E_OpStep.VMCAS_VENTING: // Venting, increase opening by X% every 2 miniutes, until at atmosphere
    DREAM_ROUGH2_VFV_02.M_SetControlMode(E_VCN.ManualControl); // set manual mode for VFV valve
    DREAM_ROUGH2_VFV_03.M_SetControlMode(E_VCN.ManualControl); // set manual mode for VFV valve
    // Verify ATM_PRESS_ERR_RNG value with testing
    IF NOT (ABS(ATM_PRESS - DREAM_DP1_GPI_01.PG.rPRESS) <= ATM_PRESS_ERR_RNG)
        AND NOT (ABS(ATM_PRESS - DREAM_MC_GPI_01.PG.rPRESS) <= ATM_PRESS_ERR_RNG)
        AND NOT (ABS(ATM_PRESS - DREAM_ROUGH2_GPI_02.PG.rPRESS) <= ATM_PRESS_ERR_RNG)
        AND NOT (ABS(ATM_PRESS - DREAM_ROUGH2_GPI_03.PG.rPRESS) <= ATM_PRESS_ERR_RNG)
    THEN
        M_RunTimeoutTimer(VENTING_CYCLE);
        M_SetMessage('Venting Started');
        // Add check if serial communication is ok. If not ok we should only stick to change open position by 1% until venting completed?
        // I think we should add range here for the speed 1-5 Hz? I think sometimes speed doesn't go all the way to 0 Hz, verify with testing
        IF M_TimeoutExpired() THEN
            M_ResetTimeoutTimer(); // Reset timer for next 2 min venting cycle
            IF (NOT (DREAM_DP1_PTM_01.iq_stPTM.i_diCurSpd < 1) OR fbSerialLineControl_DREAM_DP1_PTM_01.Error)
                AND (NOT (DREAM_DP2_PTM_01.iq_stPTM.i_diCurSpd < 1) OR fbSerialLineControl_DREAM_DP2_PTM_01.Error)
                AND (NOT (DREAM_DP3_PTM_01.iq_stPTM.i_diCurSpd < 1) OR fbSerialLineControl_DREAM_DP3_PTM_01.Error)
                AND (NOT (DREAM_MC_PTM_01.iq_stPTM.i_diCurSpd < 1) OR fbSerialLineControl_DREAM_MC_PTM_01.Error)
                AND (NOT (DREAM_MC_PTM_02.iq_stPTM.i_diCurSpd < 1) OR fbSerialLineControl_DREAM_MC_PTM_01.Error)
                AND (NOT (DREAM_CAT1_PTM_01.iq_stPTM.i_diCurSpd < 1) OR fbSerialLineControl_DREAM_CAT1_PTM_01.Error)
                AND (NOT (DREAM_CAT2_PTM_01.iq_stPTM.i_diCurSpd < 1) OR fbSerialLineControl_DREAM_CAT2_PTM_01.Error)
                AND (NOT (DREAM_ROUGH2_PTM_01.iq_stPTM.i_diCurSpd < 1) OR fbSerialLineControl_DREAM_ROUGH2_PTM_01.Error)
                AND (NOT (DREAM_ROUGH2_PTM_02.iq_stPTM.i_diCurSpd < 1) OR fbSerialLineControl_DREAM_ROUGH2_PTM_02.Error)
            THEN
                IF fRough2VFV2Position < VFV_MAX_POSITION THEN
                    fRough2VFV2Position := fRough2VFV2Position + VFV_POSITION_STEP; // every 2 min increase open positon for 1% while pumps above 1 HZ
                ELSE
                    fRough2VFV2Position := VFV_MAX_POSITION;
                END_IF

                IF fRough2VFV3Position < VFV_MAX_POSITION THEN
                    fRough2VFV3Position := fRough2VFV3Position + VFV_POSITION_STEP; // every 2 min increase open positon for 1% while pumps above 1 HZ
                ELSE
                    fRough2VFV3Position := VFV_MAX_POSITION;
                END_IF
            ELSE
                fRough2VFV2Position := VFV_MAX_POSITION; // open venting valve to max postion when pump speed reached below 1Hz
                fRough2VFV3Position := VFV_MAX_POSITION; // open venting valve to max postion when pump speed reached below 1Hz
            END_IF
        END_IF
    ELSE
        M_SetMessage('Venting completed');
        M_ResetTimeoutTimer();
        eStep := E_OpStep.VMCAS_FINISH;
    END_IF

    DREAM_ROUGH2_VFV_02.M_SetReqPosition(fRough2VFV2Position); // set venting valve position
    DREAM_ROUGH2_VFV_03.M_SetReqPosition(fRough2VFV3Position); // set venting valve position

E_OpStep.VMCAS_FINISH: // Finish procedure, close venting valves, reset set points for all valves, pumps etc.
    DREAM_ROUGH2_VFV_02.M_SetControlMode(E_VCN.CloseValve);
    DREAM_ROUGH2_VFV_03.M_SetControlMode(E_VCN.CloseValve);
    // Reset vent valve postions
    fRough2VFV2Position := 0;
    fRough2VFV3Position := 0;

    // Set the at vacuum interlocks so user can't just start opening the valves
    DREAM_ROUGH2_VRC_01.M_SetAtVacSP(VALVE_INTERLOCK_SP);
    DREAM_ROUGH2_VRC_02.M_SetAtVacSP(VALVE_INTERLOCK_SP);

    // Set the at vacuum interlocks so user can't just start turning on pumps
    DREAM_DP1_PTM_01.M_SetBackingSP(PTM_INTERLOCK_SP);
    DREAM_DP2_PTM_01.M_SetBackingSP(PTM_INTERLOCK_SP);
    DREAM_DP3_PTM_01.M_SetBackingSP(PTM_INTERLOCK_SP);
    DREAM_MC_PTM_01.M_SetBackingSP(PTM_INTERLOCK_SP);
    DREAM_MC_PTM_02.M_SetBackingSP(PTM_INTERLOCK_SP);
    DREAM_CAT1_PTM_01.M_SetBackingSP(PTM_INTERLOCK_SP);
    DREAM_CAT2_PTM_01.M_SetBackingSP(PTM_INTERLOCK_SP);
    DREAM_ROUGH2_PTM_01.M_SetBackingSP(PTM_INTERLOCK_SP);
    DREAM_ROUGH2_PTM_02.M_SetBackingSP(PTM_INTERLOCK_SP);

    // Remove command to close beamline window valves
    GVL_PLC_Interface.bCLOSE_TMO_MR5K4_VWC := FALSE;
    GVL_PLC_Interface.bCLOSE_TMO_TM2K4_VWC := FALSE;

    M_Finish();

ELSE
    M_FatalError('Operation is in invalid state');
END_CASE

END_FUNCTION_BLOCK

// ---- POUs/Automation/Abstracts/FB_Operation.TcPOU
FUNCTION_BLOCK FB_Operation
VAR_INPUT
    i_bExecute : BOOL; // Flag that indicates the operation should be ran
    i_bCancel : BOOL; // Cancel operation input signal
END_VAR
VAR_IN_OUT
    iq_sMessageBuffer : STRING(EPICS_STRING_SIZE); // Human readable description of the current step
END_VAR
VAR_OUTPUT
    q_bError : BOOL; // Whether a fatal error was encountered
    q_bBusy : BOOL; // Whether the current operation is executing
END_VAR
VAR
    bCancel : BOOL; // Saved cancel operation signal
    bDeferCancel : BOOL; // Setting to True prevents operation from being immediatly cancelled with i_bCancel. Resets to FALSE after operation finishes
    eStep : E_OpStep := E_OpStep.IDLE; // The current operation step
    fbTimeoutTimer : TON; // Timer used for tracking operation timeouts
END_VAR

IF eStep = E_OpStep.IDLE AND i_bExecute = TRUE THEN
    // Start operation
    eStep := E_OpStep.START;
    q_bBusy := TRUE;
    M_ResetError();
END_IF

(* Save the input i_bCancel signal since cancelling can take multiple cycles *)
IF i_bCancel THEN
    bCancel := TRUE;
END_IF

(* Allow operation to be cancelled from an input signal.
 The cancel input signal can be deferred by the operation if the
 operation is not at a good point to finish cancelling. *)
IF eStep <> E_OpStep.IDLE AND NOT bDeferCancel AND bCancel THEN
    M_Cancel();
END_IF

IF M_TimeoutExpired() THEN // If a timeout has expired, trigger a fatal error
    M_FatalError('Timeout expired');
END_IF

METHOD PROTECTED M_Cancel
VAR_INPUT
END_VAR
M_ResetTimeoutTimer();
M_SetMessage('Operation canceled');
eStep := E_OpStep.IDLE;
q_bBusy := FALSE;
bCancel := FALSE;
M_DeferCancel(FALSE);
END_METHOD

// Defer cancel signals until a later time
METHOD PROTECTED M_DeferCancel
VAR_INPUT
    i_bDefer : BOOL;
END_VAR
bDeferCancel := i_bDefer;
END_METHOD

METHOD PROTECTED M_FatalError
VAR_INPUT
    i_ErrorMessage : STRING;
END_VAR
M_ResetTimeoutTimer();
M_SetMessage(i_ErrorMessage);
eStep := E_OpStep.IDLE;
q_bError := TRUE;
q_bBusy := FALSE;
bCancel := FALSE;
M_DeferCancel(FALSE);
END_METHOD

METHOD PROTECTED M_Finish
VAR_INPUT
END_VAR
M_ResetTimeoutTimer();
M_SetMessage('Operation finished');
eStep := E_OpStep.IDLE;
q_bBusy := FALSE;
bCancel := FALSE;
M_DeferCancel(FALSE);
END_METHOD

METHOD PROTECTED M_ResetError
VAR_INPUT
END_VAR
q_bError := FALSE;
END_METHOD

METHOD PROTECTED M_ResetTimeoutTimer
VAR_INPUT
END_VAR
fbTimeoutTimer(IN := FALSE);
END_METHOD

METHOD PROTECTED M_RunTimeoutTimer
VAR_INPUT
    i_tTime : TIME; // How long the timer should run before signalling a timeout
END_VAR
fbTimeoutTimer(IN := TRUE, PT := i_tTime);
END_METHOD

METHOD PROTECTED M_SetMessage
VAR_INPUT
    i_sMessage : STRING(EPICS_STRING_SIZE);
END_VAR
iq_sMessageBuffer := i_sMessage;
END_METHOD

METHOD PROTECTED M_TimeoutExpired : BOOL
VAR_INPUT
END_VAR
fbTimeoutTimer(); // Advance timer
M_TimeoutExpired := fbTimeoutTimer.Q;
END_METHOD

END_FUNCTION_BLOCK

// ---- POUs/Automation/FB_AtVacuum.TcPOU
FUNCTION_BLOCK FB_AtVacuum EXTENDS FB_Operation
VAR_INPUT
END_VAR
VAR_OUTPUT
END_VAR
VAR
END_VAR

SUPER^(iq_sMessageBuffer := iq_sMessageBuffer);

CASE eStep OF
E_OpStep.IDLE: // Do nothing

E_OpStep.START: // Start monitoring main chamber vacuum
    IF NOT (F_AllPumpsRunning() AND F_PressAtVacSP()) THEN // add case if already vented to just cancel operation
        M_RunTimeoutTimer(TURBOS_NOT_RUNNING_TIMEOUT);
        M_SetMessage('Vacuum lost, 10 min timer started');
        IF M_TimeoutExpired() THEN
            M_FatalError('Vacuum not restored, venting started');
        END_IF
    ELSE
        M_ResetTimeoutTimer(); //reset timer if pump restarted or gauge restarted and vaccum ok
        M_SetMessage('MC Vacuum OK');
    END_IF

ELSE
    M_FatalError('Operation is in invalid state');
END_CASE

END_FUNCTION_BLOCK

// ---- POUs/Functions/F_AllPumpsRunning.TcPOU
FUNCTION F_AllPumpsRunning : BOOL
VAR_INPUT
END_VAR
VAR
END_VAR

// Pump running state verifys that iq_stPtm.i_xAtSpd AND iq_stPtm.q_RunDO are TRUE
F_AllPumpsRunning := //DREAM_NC_PTM_01.iq_stPTM.eState = E_PumpState.pumpRUNNING AND
                     //DREAM_NC_PTM_02.iq_stPTM.eState = E_PumpState.pumpRUNNING AND
                     DREAM_DP1_PTM_01.iq_stPTM.eState = E_PumpState.pumpRUNNING AND
                     DREAM_DP2_PTM_01.iq_stPTM.eState = E_PumpState.pumpRUNNING AND
                     DREAM_DP3_PTM_01.iq_stPTM.eState = E_PumpState.pumpRUNNING AND
                     DREAM_MC_PTM_01.iq_stPTM.eState = E_PumpState.pumpRUNNING AND
                     DREAM_MC_PTM_02.iq_stPTM.eState = E_PumpState.pumpRUNNING AND
                     DREAM_CAT1_PTM_01.iq_stPTM.eState = E_PumpState.pumpRUNNING AND
                     DREAM_CAT2_PTM_01.iq_stPTM.eState = E_PumpState.pumpRUNNING AND
                     DREAM_ROUGH2_PTM_01.iq_stPTM.eState = E_PumpState.pumpRUNNING AND
                     DREAM_ROUGH2_PTM_02.iq_stPTM.eState = E_PumpState.pumpRUNNING;

END_FUNCTION

// ---- POUs/Functions/F_PressAtVacSP.TcPOU
FUNCTION F_PressAtVacSP : BOOL
VAR_INPUT
END_VAR
VAR
END_VAR

F_PressAtVacSP := //DREAM_NC_GCC_01.IG.rPRESS < ATVAC_INTERLOCK_SP AND DREAM_NC_GCC_01.IG.xPRESS_OK AND
                  //DREAM_DP1_GHC_01.IG.rPRESS < ATVAC_INTERLOCK_SP AND DREAM_DP1_GHC_01.IG.xPRESS_OK AND
                  //DREAM_DP2_GHC_01.IG.rPRESS < ATVAC_INTERLOCK_SP AND DREAM_DP2_GHC_01.IG.xPRESS_OK AND
                  //DREAM_DP3_GHC_01.IG.rPRESS < ATVAC_INTERLOCK_SP AND DREAM_DP3_GHC_01.IG.xPRESS_OK AND
                  //DREAM_CAT1_GHC_01.IG.rPRESS < ATVAC_INTERLOCK_SP AND DREAM_CAT1_GHC_01.IG.xPRESS_OK AND
                  //DREAM_CAT2_GHC_01.IG.rPRESS < ATVAC_INTERLOCK_SP AND DREAM_CAT2_GHC_01.IG.xPRESS_OK AND
                  GVL_VAC_GAUGES.stDREAM_MC_GAUGE.rPRESS < AT_VAC_SP AND GVL_VAC_GAUGES.stDREAM_MC_GAUGE.xPRESS_OK;
                  //GVL_VAC_GAUGES.stDREAM_MC_GHC.xAT_VAC;
                  //we could also be checking ST_VG.xAT_VAC flag and make this value changeable?

END_FUNCTION

// ---- POUs/Functions/F_IsValidStateTransition.TcPOU
FUNCTION F_IsValidStateTransition : BOOL
VAR_INPUT
    eCurrentState : E_Op;
    eNextState : E_Op;
END_VAR
VAR
END_VAR

CASE eCurrentState OF

E_Op.INIT:
    F_IsValidStateTransition := (eNextState = E_Op.STANDBY);

E_Op.STANDBY:
    F_IsValidStateTransition := (eNextState = E_Op.STANDBY) OR
                                //(eNextState = E_Op.PUMP_ALL) OR
                                //(eNextState = E_Op.PUMP_NC) OR
                                (eNextState = E_Op.VENT_MC_CAT); // OR
                                //(eNextState = E_Op.VENT_ALL) OR
                                //(eNextState = E_Op.VENT_NC) OR
                                //(eNextState = E_Op.VENT_CAT);
                                //uncomment after procedures implemented
E_Op.PUMP_ALL:
    F_IsValidStateTransition := (eNextState = E_Op.STANDBY);

E_Op.PUMP_NC:
    F_IsValidStateTransition := (eNextState = E_Op.STANDBY);

E_Op.AT_VACUUM:
    F_IsValidStateTransition := (eNextState = E_Op.VENT_MC_CAT); //OR
                                //(eNextState = E_Op.VENT_ALL) OR
                                //(eNextState = E_Op.VENT_NC) OR
                                //(eNextState = E_Op.VENT_CAT);
                                //uncomment after procedures implemented

E_Op.VENT_ALL:
    F_IsValidStateTransition := (eNextState = E_Op.STANDBY);

E_Op.VENT_NC:
    F_IsValidStateTransition := (eNextState = E_Op.STANDBY);

E_Op.VENT_MC_CAT:
    F_IsValidStateTransition := (eNextState = E_Op.STANDBY);

E_Op.VENT_CAT:
    F_IsValidStateTransition := (eNextState = E_Op.STANDBY);

ELSE
    F_IsValidStateTransition := FALSE;
END_CASE;

END_FUNCTION

// ---- POUs/PRG_COM.TcPOU
PROGRAM PRG_COM
VAR

END_VAR

(*Instanitate Serial port com function *)
fbSerialLineControl_DREAM_NC_PTM_01(
    Mode:= SERIALLINEMODE_EL6_22B,
    pComIn:= ADR(stComIn_DREAM_NC_PTM_01),
    pComOut:= ADR(stComOut_DREAM_NC_PTM_01),
    SizeComIn:= UINT_TO_INT(SIZEOF(stComIn_DREAM_NC_PTM_01)),
    TxBuffer:= SerialTXBuffer_DREAM_NC_PTM_01,
    RxBuffer:= SerialRXBuffer_DREAM_NC_PTM_01,
    Error=> ,
    ErrorID=> );

fbSerialLineControl_DREAM_NC_PTM_02(
    Mode:= SERIALLINEMODE_EL6_22B,
    pComIn:= ADR(stComIn_DREAM_NC_PTM_02),
    pComOut:= ADR(stComOut_DREAM_NC_PTM_02),
    SizeComIn:= UINT_TO_INT(SIZEOF(stComIn_DREAM_NC_PTM_02)),
    TxBuffer:= SerialTXBuffer_DREAM_NC_PTM_02,
    RxBuffer:= SerialRXBuffer_DREAM_NC_PTM_02,
    Error=> ,
    ErrorID=> );

fbSerialLineControl_DREAM_DP1_PTM_01(
    Mode:= SERIALLINEMODE_EL6_22B,
    pComIn:= ADR(stComIn_DREAM_DP1_PTM_01),
    pComOut:= ADR(stComOut_DREAM_DP1_PTM_01),
    SizeComIn:= UINT_TO_INT(SIZEOF(stComIn_DREAM_DP1_PTM_01)),
    TxBuffer:= SerialTXBuffer_DREAM_DP1_PTM_01,
    RxBuffer:= SerialRXBuffer_DREAM_DP1_PTM_01,
    Error=> ,
    ErrorID=> );

fbSerialLineControl_DREAM_DP2_PTM_01(
    Mode:= SERIALLINEMODE_EL6_22B,
    pComIn:= ADR(stComIn_DREAM_DP2_PTM_01),
    pComOut:= ADR(stComOut_DREAM_DP2_PTM_01),
    SizeComIn:= UINT_TO_INT(SIZEOF(stComIn_DREAM_DP2_PTM_01)),
    TxBuffer:= SerialTXBuffer_DREAM_DP2_PTM_01,
    RxBuffer:= SerialRXBuffer_DREAM_DP2_PTM_01,
    Error=> ,
    ErrorID=> );

fbSerialLineControl_DREAM_DP3_PTM_01(
    Mode:= SERIALLINEMODE_EL6_22B,
    pComIn:= ADR(stComIn_DREAM_DP3_PTM_01),
    pComOut:= ADR(stComOut_DREAM_DP3_PTM_01),
    SizeComIn:= UINT_TO_INT(SIZEOF(stComIn_DREAM_DP3_PTM_01)),
    TxBuffer:= SerialTXBuffer_DREAM_DP3_PTM_01,
    RxBuffer:= SerialRXBuffer_DREAM_DP3_PTM_01,
    Error=> ,
    ErrorID=> );

fbSerialLineControl_DREAM_MC_PTM_01(
    Mode:= SERIALLINEMODE_EL6_22B,
    pComIn:= ADR(stComIn_DREAM_MC_PTM_01),
    pComOut:= ADR(stComOut_DREAM_MC_PTM_01),
    SizeComIn:= UINT_TO_INT(SIZEOF(stComIn_DREAM_MC_PTM_01)),
    TxBuffer:= SerialTXBuffer_DREAM_MC_PTM_01,
    RxBuffer:= SerialRXBuffer_DREAM_MC_PTM_01,
    Error=> ,
    ErrorID=> );

fbSerialLineControl_DREAM_MC_PTM_02(
    Mode:= SERIALLINEMODE_EL6_22B,
    pComIn:= ADR(stComIn_DREAM_MC_PTM_02),
    pComOut:= ADR(stComOut_DREAM_MC_PTM_02),
    SizeComIn:= UINT_TO_INT(SIZEOF(stComIn_DREAM_MC_PTM_02)),
    TxBuffer:= SerialTXBuffer_DREAM_MC_PTM_02,
    RxBuffer:= SerialRXBuffer_DREAM_MC_PTM_02,
    Error=> ,
    ErrorID=> );

fbSerialLineControl_DREAM_CAT1_PTM_01(
    Mode:= SERIALLINEMODE_EL6_22B,
    pComIn:= ADR(stComIn_DREAM_CAT1_PTM_01),
    pComOut:= ADR(stComOut_DREAM_CAT1_PTM_01),
    SizeComIn:= UINT_TO_INT(SIZEOF(stComIn_DREAM_CAT1_PTM_01)),
    TxBuffer:= SerialTXBuffer_DREAM_CAT1_PTM_01,
    RxBuffer:= SerialRXBuffer_DREAM_CAT1_PTM_01,
    Error=> ,
    ErrorID=> );

fbSerialLineControl_DREAM_CAT2_PTM_01(
    Mode:= SERIALLINEMODE_EL6_22B,
    pComIn:= ADR(stComIn_DREAM_CAT2_PTM_01),
    pComOut:= ADR(stComOut_DREAM_CAT2_PTM_01),
    SizeComIn:= UINT_TO_INT(SIZEOF(stComIn_DREAM_CAT2_PTM_01)),
    TxBuffer:= SerialTXBuffer_DREAM_CAT2_PTM_01,
    RxBuffer:= SerialRXBuffer_DREAM_CAT2_PTM_01,
    Error=> ,
    ErrorID=> );

fbSerialLineControl_DREAM_ROUGH2_PTM_01(
    Mode:= SERIALLINEMODE_EL6_22B,
    pComIn:= ADR(stComIn_DREAM_ROUGH2_PTM_01),
    pComOut:= ADR(stComOut_DREAM_ROUGH2_PTM_01),
    SizeComIn:= UINT_TO_INT(SIZEOF(stComIn_DREAM_ROUGH2_PTM_01)),
    TxBuffer:= SerialTXBuffer_DREAM_ROUGH2_PTM_01,
    RxBuffer:= SerialRXBuffer_DREAM_ROUGH2_PTM_01,
    Error=> ,
    ErrorID=> );

fbSerialLineControl_DREAM_ROUGH2_PTM_02(
    Mode:= SERIALLINEMODE_EL6_22B,
    pComIn:= ADR(stComIn_DREAM_ROUGH2_PTM_02),
    pComOut:= ADR(stComOut_DREAM_ROUGH2_PTM_02),
    SizeComIn:= UINT_TO_INT(SIZEOF(stComIn_DREAM_ROUGH2_PTM_02)),
    TxBuffer:= SerialTXBuffer_DREAM_ROUGH2_PTM_02,
    RxBuffer:= SerialRXBuffer_DREAM_ROUGH2_PTM_02,
    Error=> ,
    ErrorID=> );

END_PROGRAM

// ---- POUs/Functions/F_TurboIlkLogic.TcPOU
FUNCTION F_TurboIlkLogic : BOOL
VAR_INPUT
    i_stTurbo : ST_PTM; //Turbo Pump
    //i_stISG : ST_VG; //Gauge measuring inlet Pressure e.g Pirani
    i_stBackingGauge : ST_VG; //Gauge measuring backing pressure
    i_stRoughValve : ST_VGC; //Roughing Valve on the turbo pump backing line
END_VAR
VAR
END_VAR

F_TurboIlkLogic := i_stBackingGauge.rPRESS < i_stTurbo.rBackingPressureSP AND i_stBackingGauge.xPRESS_OK AND
                   i_stRoughValve.i_xOpnLS;

END_FUNCTION
